INTERFACE INTERNAL I_TagCmp

METHOD AndIf : I_TagCmp
VAR_INPUT
	bCondition: BOOL;
END_VAR
END_METHOD

METHOD Default : BOOL
END_METHOD

METHOD IsErr : BOOL
END_METHOD

METHOD IsOk : BOOL
END_METHOD

METHOD Match : I_TagCmp
VAR_INPUT
	iOther: I_Tag;
END_VAR
END_METHOD

METHOD MatchId : I_TagCmp
VAR_INPUT
	sOtherId	: Strings.Str;
END_VAR
END_METHOD

METHOD MatchPrtId : I_TagCmp
VAR_INPUT
	sPartialId		: Strings.Str;
END_VAR
END_METHOD

METHOD OrIf : I_TagCmp
VAR_INPUT
	bCondition: BOOL;
END_VAR
END_METHOD

METHOD Set : I_TagCmp
VAR_INPUT
	iBaseTag	: I_Tag;
END_VAR
END_METHOD

METHOD XorIf : I_TagCmp
VAR_INPUT
	bCondition: BOOL;
END_VAR
END_METHOD

END_INTERFACE

(* stored: Version 1.1.0.1
   Itf I_TagCmp: Id {434164ab-6703-48fd-8c7c-cbf390d14597}
   Method AndIf: Id {436de305-153d-45a1-9c24-e403a9752ee1}
   Method Default: Id {49b183b3-7ff3-4c1f-86ad-ab7ad18768ea}
   Method IsErr: Id {bdea08ea-65d7-4af4-a4f6-f3da4269e7d0}
   Method IsOk: Id {9e31c3a1-a234-461e-97b6-7c042a50360a}
   Method Match: Id {ff272183-aeae-424d-9c25-2144ef81905e}
   Method MatchId: Id {68b43ba9-4c50-40a8-b666-e36aaf6996e2}
   Method MatchPrtId: Id {5cba49aa-7253-4bc9-829c-d83e4b3c65d2}
   Method OrIf: Id {43b0b3b9-ad9a-4aeb-88cb-22e31aac3fe8}
   Method Set: Id {94ae1389-8107-4a7f-b005-7ced5ba44f46}
   Method XorIf: Id {d8e35498-785d-4895-9e65-30990ff7fe09} *)
